{attribute 'linkalways'} 
{attribute 'no_explicit_call' := 'This FB is a CLASS and must be accessed using methods or properties'}
{attribute 'enable_dynamic_creation'}
FUNCTION_BLOCK INTERNAL MoveRelativeCommand EXTENDS MoveCommand
VAR
	_fb : MC_MoveRelative;
	_distance : LREAL;
END_VAR

METHOD FB_init : BOOL
VAR_INPUT
	bInitRetains : BOOL; // if TRUE, the retain variables are initialized (warm start / cold start)
	bInCopyCode : BOOL;  // if TRUE, the instance afterwards gets moved into the copy code (online change)
	axisRef : REFERENCE TO Axis;
	distance : LREAL;
	velocity : LREAL;
	acceleration : LREAL;
	deceleration : LREAL;
	jerk : LREAL;
	bufferMode : AxisBufferMode;
END_VAR
_axisRef REF= axisRef;
_distance := distance;
_velocity := velocity;
_acceleration := acceleration;
_deceleration := deceleration;
_jerk := jerk;
_bufferMode := bufferMode;
END_METHOD

METHOD PROTECTED WhileBusy
VAR_INPUT
	CommandState : I_CommandBusyState;
END_VAR
_fb(
	Axis := _axisRef._InternalAxisRef,
	Execute := TRUE,
	Distance := _distance,
	Velocity := _velocity,
	Acceleration := _acceleration,
	Deceleration := _deceleration,
	Jerk := _jerk,
	BufferMode := _bufferMode
);

IF _fb.Busy THEN
	RETURN;
END_IF

IF _fb.CommandAborted THEN
	_fb(Axis := _axisRef._InternalAxisRef, Execute := FALSE);
	CommandState.SetAborting();
	RETURN;
END_IF

IF _fb.Error THEN
	_fb(Axis := _axisRef._InternalAxisRef, Execute := FALSE);
	CommandState.SetError(_fb.ErrorID);
	RETURN;
END_IF

_fb(Axis := _axisRef._InternalAxisRef, Execute := FALSE);
CommandState.SetDone();
END_METHOD

END_FUNCTION_BLOCK

(* stored: Version 1.1.0.1, ProductVersion 3.1.4024.12
   POU MoveRelativeCommand: Id {0489af38-80cf-48c1-b1e3-c03536e8b586}, SpecialFunc None
   Folder Constructor: Id {0880fa7c-2919-4030-88be-790fc93e651a}
   Method FB_init: Id {b5d5a662-7f77-4804-aaf2-75cbd9df0dea}
   Method WhileBusy: Id {0d6e5cfe-9804-4418-8f36-9ae6df55ae3f} *)
